// TIA Portal V17 export
// export: Created 2023-02-13T11:16:46.229804Z, ExportSetting WithDefaults, DisplayName Totally Integrated Automation Portal, DisplayVersion V17, DisplayName TIA Portal Openness, DisplayVersion V17, DisplayName TIA Portal Teamcenter Gateway, DisplayVersion V17, DisplayName TIA Portal Version Control Interface, DisplayVersion V17, DisplayName SINAMICS Startdrive Advanced, DisplayVersion V17, DisplayName SINAMICS Startdrive G130, G150, S120, S150, SINAMICS MV, S210, DisplayVersion V17, DisplayName SINAMICS Startdrive G110M, G120, G120C, G120D, G120P, G115D, DisplayVersion V17, DisplayName STEP 7 Professional, DisplayVersion V17, DisplayName STEP 7 Safety, DisplayVersion V17, DisplayName WinCC Professional, DisplayVersion V17
DATA_BLOCK "General_DB"   // DB47
{ S7_Optimized_Access := 'TRUE' }
VERSION : 0.1
// stored: AutoNumber false, DBAccessibleFromOPCUA true, DBAccessibleFromWebserver true, IsOnlyStoredInLoadMemory false, IsRetainMemResEnabled false, IsWriteProtectedInAS false, MemoryReserve 100
   VAR
      Initial : Bool;
      "Reset HMI Prep" : Bool;
      "Reset HMI ST" : Bool;
      "Reset HMI Blend" : Bool;
      "Reset Scada" : Bool;
      Reset : Bool;
      Reset_Dose : Bool;
      Sim_Mode : Bool;   // 1 Simulation
      Sim_ON : Bool;
      Sim_OFF : Bool;
      Man_Initi : Bool;
      LDT_PLC : Date_And_Time;
      LDT_retval : Int;
      CIP_Line1_Open : Struct
         "CIP Tank_T01" : Bool;
         "CIP Line_T01" : Bool;
         "CIP Tank_T02" : Bool;
         "CIP Line_T02" : Bool;
         "CIP Tank_T03" : Bool;
         "CIP Line_T03" : Bool;
         "CIP Tank_T04" : Bool;
         "CIP Line_T04" : Bool;
         "CIP Tank_T05" : Bool;
         "CIP Line_T05" : Bool;
         "CIP Tank_T06" : Bool;
         "CIP Line_T06" : Bool;
         "CIP Tank_T07" : Bool;
         "CIP Line_T07" : Bool;
         "CIP Tank_T08" : Bool;
         "CIP Line_T08" : Bool;
         "CIP Tank_T09" : Bool;
         "CIP Line_T09" : Bool;
         "CIP Tank_T10" : Bool;
         "CIP Line_T10" : Bool;
         "CIP Tank_T11" : Bool;
         "CIP Line_T11" : Bool;
         "CIP Tank_T12" : Bool;
         "CIP Line_T12" : Bool;
         "CIP Tank_T13" : Bool;
         "CIP Line_T13" : Bool;
         CIP_Tank : Bool;
         CIP_Line : Bool;
      END_STRUCT;
      CIP_Line2_Open : Struct
         "CIP Tank_T1" : Bool;
         "CIP Line_T1" : Bool;
         "CIP Tank_T2" : Bool;
         "CIP Line_T2" : Bool;
         "CIP Tank_T3" : Bool;
         "CIP Line_T3" : Bool;
         "CIP Tank_T4" : Bool;
         "CIP Line_T4" : Bool;
         "CIP Tank_T5" : Bool;
         "CIP Line_T5" : Bool;
         "CIP Tank_T6" : Bool;
         "CIP Line_T6" : Bool;
         "CIP Tank_T7" : Bool;
         "CIP Line_T7" : Bool;
         "CIP Tank_T8" : Bool;
         "CIP Line_T8" : Bool;
         "CIP Tank_T9" : Bool;
         "CIP Line_T9" : Bool;
         "CIP Tank_T10" : Bool;
         "CIP Line_T10" : Bool;
         CIP_Tank : Bool;
         CIP_Line : Bool;
      END_STRUCT;
      "Bypass CIP Signal Storage" : Bool;
      "Bypass CIP Signal Homomixer" : Bool;
      "Testing FB Valve" : Struct
         Preparation : Bool;
         Homomixer : Bool;
         Blending : Bool;
         Storage : Bool;
      END_STRUCT;
      "Testing FB Motor" : Struct
         "MCC Blending" : Bool;
         "MCC Preparation" : Bool;
      END_STRUCT;
      "CIP Drain Time" : Struct
         BlendingCluster1 : TOF_TIME;
         BlendingCluster2 : TOF_TIME;
         "Preparation_02.20" : TOF_TIME;
         "Preparation_05.20" : TOF_TIME;
         Homomixer : TOF_TIME;
         "Storage_29.06" : TOF_TIME;
         "Storage_39.06" : TOF_TIME;
         HMI_Input : Struct
            BlendingCluster1 : Int := 60;
            BlendingCluster2 : Int := 60;
            "Preparation_02.20" : Int := 60;
            "Preparation_05.20" : Int := 60;
            Homomixer : Int := 60;
            "Storage_29.06" : Int := 60;
            "Storage_39.06" : Int := 60;
         END_STRUCT;
         Actual : Struct
            BlendingCluster1 : DInt;
            BlendingCluster2 : DInt;
            "Preparation_02.20" : DInt;
            "Preparation_05.20" : DInt;
            Homomixer : DInt;
            "Storage_29.06" : DInt;
            "Storage_39.06" : DInt;
         END_STRUCT;
      END_STRUCT;
   END_VAR
BEGIN
   "CIP Drain Time".BlendingCluster1.PT := T#1m;
   "CIP Drain Time".BlendingCluster2.PT := T#1m;
   "CIP Drain Time"."Preparation_02.20".PT := T#1m;
   "CIP Drain Time"."Preparation_05.20".PT := T#1m;
   "CIP Drain Time".Homomixer.PT := T#1m;
   "CIP Drain Time"."Storage_29.06".PT := T#1m;
   "CIP Drain Time"."Storage_39.06".PT := T#1m;
END_DATA_BLOCK
